// TIA Portal V19 export
DATA_BLOCK "AreaGen_Messages"   // DB179
// stored: MemoryReserve 100
   VAR
      "A" : Struct
         Msg : Array[1..304] of Bool;
         Hmi : Array[1..19] of Word;
         Ack : Array[1..19] of Word;
      END_STRUCT;
      W : Struct
         Msg : Array[1..256] of Bool;
         Hmi : Array[1..16] of Word;
         Ack : Array[1..16] of Word;
      END_STRUCT;
      Area01_A_Counter : Int;
      Area01_W_Counter : Int;
      Area02_A_Counter : Int;
      Area02_W_Counter : Int;
      Area03_A_Counter : Int;
      Area03_W_Counter : Int;
   END_VAR
BEGIN
   // "A".Msg[2] : h
   // "A".Msg[3] : hsfdd
   // W.Msg[2] : h
   // W.Msg[3] : hsfdd
END_DATA_BLOCK
